// TIA Portal project "OPCUA_CLIENT" (V17)

(* hardware
DEVICE "S7-1500/ET200MP station_1"  S7-1500 station
   slot 0: "Rail_0"  Rack  6ES7 590-1***0-0AA0
   slot 1: "OPC_CLIENT"  CPU 1511-1 PN  6ES7 511-1AK01-0AB0  V2.8
      slot 3: "CPU display_1"  6ES7591-1AA00-0AA0
      slot 32768: "PROFINET interface_1"  X1
         slot 32769: "Port_1"  X1 P1
         slot 32770: "Port_2"  X1 P2
      slot 34817: "Virtual CP interface port_1"  Virtual CP interface port  Virtual CP interface port
*)

// ===== PLC "OPC_CLIENT"  CPU 1511-1 PN =====

VAR_GLOBAL   // PLC tag table "Default tag table"
   "DISCONECT" AT %M201.0 : Bool;
   "Tag_1" AT %M201.1 : Bool;
   "Tag_2" AT %M102.0 : Bool;
   "Tag_3" AT %M100.0 : Bool;
   "GetNameSpace" AT %M100.1 : Bool;
   "GetNodeHandleList" AT %M0.0 : Bool;
   "Clock_Byte" AT %MB10 : Byte;
   "Clock_10Hz" AT %M10.0 : Bool;
   "Clock_5Hz" AT %M10.1 : Bool;
   "Clock_2.5Hz" AT %M10.2 : Bool;
   "Clock_2Hz" AT %M10.3 : Bool;
   "Clock_1.25Hz" AT %M10.4 : Bool;
   "Clock_1Hz" AT %M10.5 : Bool;
   "Clock_0.625Hz" AT %M10.6 : Bool;
   "Clock_0.5Hz" AT %M10.7 : Bool;
END_VAR

// folder: SystemDataTypeFolder

TYPE "Client interface_1.Read list_1"
   STRUCT
      LEVEL : Int;
      PRESSURE : Int;
   END_STRUCT;
END_TYPE

// folder: (top level)

DATA_BLOCK "Client interface_1_Data"   // DB3
{ S7_Optimized_Access := 'TRUE' }
   VAR
      "Read list_1" : Struct
         Variable : "Client interface_1.Read list_1";
         NodeStatusList : Array[0..1] of DWord;
         TimeStamps : Array[0..1] of LDT;
      END_STRUCT;
   END_VAR
BEGIN
END_DATA_BLOCK

// folder: System blocks/Program resources

DATA_BLOCK "Client interface_1_Configuration"   // DB2
{ S7_Optimized_Access := 'TRUE' }
   VAR
      Connection : Struct
         ConnectInfo : OPC_UA_SessionConnectInfo;
         ConnectionHdl : DWord;
         ServerEndpointUrl : String[254] := 'opc.tcp://192.168.100.16:4840';
      END_STRUCT;
      Namespaces : Struct
         NamespaceURIs : Array[0..0] of WString;
         ServerNamespaceIndexes : Array[0..0] of UInt;
         NamespaceStatusList : Array[0..0] of DWord;
         NamespaceCount : UInt := 1;
      END_STRUCT;
      ReadLists : Struct
         "Read list_1" : Struct
            NodeCount : UInt := 2;
            Nodes : Array[0..1] of OPC_UA_NodeId;
            NodeHdls : Array[0..1] of DWord;
         END_STRUCT;
      END_STRUCT;
   END_VAR
BEGIN
   ReadLists."Read list_1".Nodes[0].NamespaceIndex := 0;
   ReadLists."Read list_1".Nodes[0].IdentifierType := 1;
   ReadLists."Read list_1".Nodes[0].Identifier := WSTRING#'"LEVEL"';
   ReadLists."Read list_1".Nodes[1].NamespaceIndex := 0;
   ReadLists."Read list_1".Nodes[1].IdentifierType := 1;
   ReadLists."Read list_1".Nodes[1].Identifier := WSTRING#'"PRESSURE"';
   Connection.ConnectInfo.SessionName := WSTRING#'OPC UA Connection_1';
   Connection.ConnectInfo.ApplicationName := WSTRING#'';
   Connection.ConnectInfo.SecurityMsgMode := 1;
   Connection.ConnectInfo.SecurityPolicy := 1;
   Connection.ConnectInfo.CheckServerCertificate := False;
   Connection.ConnectInfo.TransportProfile := 1;
   Connection.ConnectInfo.UserIdentityTokenType := 0;
   Connection.ConnectInfo.CertificateID := 0;
   Connection.ConnectInfo.SessionTimeout := T#30S;
   Connection.ConnectInfo.MonitorConnection := T#5S;
   Connection.ConnectInfo.LocaleIDs[0] := 'en-US';
   Connection.ConnectInfo.LocaleIDs[1] := '';
   Connection.ConnectInfo.LocaleIDs[2] := '';
   Connection.ConnectInfo.LocaleIDs[3] := '';
   Connection.ConnectInfo.LocaleIDs[4] := '';
   Namespaces.NamespaceURIs[0] := WSTRING#'http://www.siemens.com/simatic-s7-opcua';
END_DATA_BLOCK

// folder: (top level)

ORGANIZATION_BLOCK "Main"   // OB1, FBD, ProgramCycle
TITLE = "Main Program Sweep (Cycle)"
{ S7_Optimized_Access := 'TRUE' }
VERSION : 0.1
   VAR_INPUT
      Initial_Call : Bool;   // Initial call of this OB
      Remanence : Bool;   // =True, if remanent data are available
   END_VAR
BEGIN

REGION Network 1
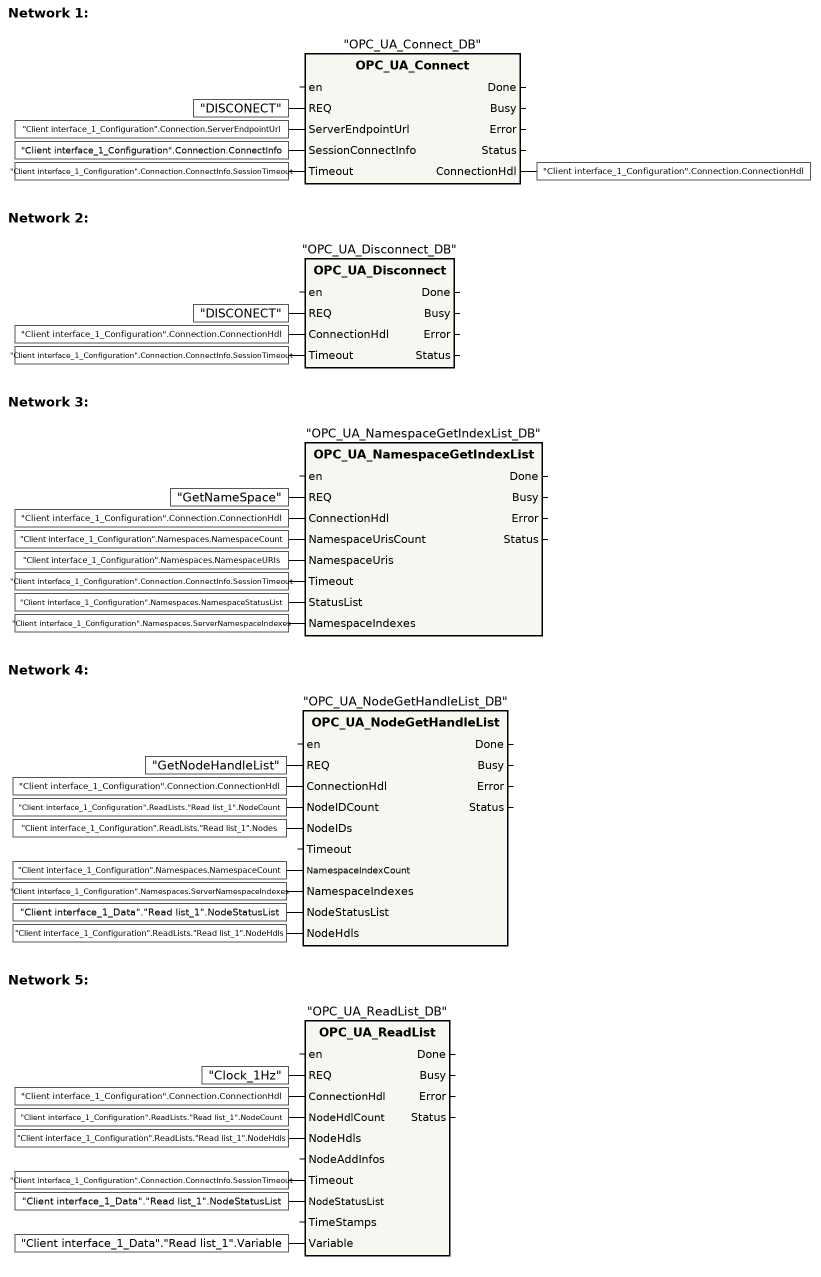
   "OPC_UA_Connect_DB"(REQ := "DISCONECT",   // OPC_UA_Connect
                       ServerEndpointUrl := "Client interface_1_Configuration".Connection.ServerEndpointUrl,
                       SessionConnectInfo := "Client interface_1_Configuration".Connection.ConnectInfo,
                       Timeout := "Client interface_1_Configuration".Connection.ConnectInfo.SessionTimeout,
                       ConnectionHdl => "Client interface_1_Configuration".Connection.ConnectionHdl);
END_REGION

REGION Network 2
   "OPC_UA_Disconnect_DB"(REQ := "DISCONECT",   // OPC_UA_Disconnect
                          ConnectionHdl := "Client interface_1_Configuration".Connection.ConnectionHdl,
                          Timeout := "Client interface_1_Configuration".Connection.ConnectInfo.SessionTimeout);
END_REGION

REGION Network 3
   "OPC_UA_NamespaceGetIndexList_DB"(REQ := "GetNameSpace",   // OPC_UA_NamespaceGetIndexList
                           ConnectionHdl := "Client interface_1_Configuration".Connection.ConnectionHdl,
                           NamespaceUrisCount := "Client interface_1_Configuration".Namespaces.NamespaceCount,
                           NamespaceUris := "Client interface_1_Configuration".Namespaces.NamespaceURIs,
                           Timeout := "Client interface_1_Configuration".Connection.ConnectInfo.SessionTimeout,
                           StatusList := "Client interface_1_Configuration".Namespaces.NamespaceStatusList,
                           NamespaceIndexes := "Client interface_1_Configuration".Namespaces.ServerNamespaceIndexes);
END_REGION

REGION Network 4
   "OPC_UA_NodeGetHandleList_DB"(REQ := "GetNodeHandleList",   // OPC_UA_NodeGetHandleList
                           ConnectionHdl := "Client interface_1_Configuration".Connection.ConnectionHdl,
                           NodeIDCount := "Client interface_1_Configuration".ReadLists."Read list_1".NodeCount,
                           NodeIDs := "Client interface_1_Configuration".ReadLists."Read list_1".Nodes,
                           NamespaceIndexCount := "Client interface_1_Configuration".Namespaces.NamespaceCount,
                           NamespaceIndexes := "Client interface_1_Configuration".Namespaces.ServerNamespaceIndexes,
                           NodeStatusList := "Client interface_1_Data"."Read list_1".NodeStatusList,
                           NodeHdls := "Client interface_1_Configuration".ReadLists."Read list_1".NodeHdls);
END_REGION

REGION Network 5
   "OPC_UA_ReadList_DB"(REQ := "Clock_1Hz",   // OPC_UA_ReadList
                        ConnectionHdl := "Client interface_1_Configuration".Connection.ConnectionHdl,
                        NodeHdlCount := "Client interface_1_Configuration".ReadLists."Read list_1".NodeCount,
                        NodeHdls := "Client interface_1_Configuration".ReadLists."Read list_1".NodeHdls,
                        Timeout := "Client interface_1_Configuration".Connection.ConnectInfo.SessionTimeout,
                        NodeStatusList := "Client interface_1_Data"."Read list_1".NodeStatusList,
                        Variable := "Client interface_1_Data"."Read list_1".Variable);
END_REGION
END_ORGANIZATION_BLOCK